TYPE T_Ctrl_SIf_JUN_Out :
STRUCT
	///switch valve retract
	bolOpen: T_Ctrl_IoBool;
END_STRUCT
END_TYPE

(* stored: Version 1.1.0.1, ProductVersion 3.1.0.23
   DUT T_Ctrl_SIf_JUN_Out: Id {97f2d690-4633-4718-8427-a5bdbe604e9a} *)
